TYPE st_NeedleActionBatch :
STRUCT
	mode			: E_mode;
	Handshake		: ST_HandshakeBase;
END_STRUCT
END_TYPE

(* stored: Version 1.1.0.1, ProductVersion 3.1.4024.13
   DUT st_NeedleActionBatch: Id {17ed98c2-5f3f-421f-b717-2ad754274d48} *)
